{attribute 'qualified_only'}
VAR_GLOBAL
    stUnknownState: DUT_PositionState := (sName := 'Unknown');
    stInvalidState: DUT_PositionState;
END_VAR

(* stored: Version 1.1.0.1, ProductVersion 3.1.4022.18
   GVL MOTION_GVL: Id {7b3cfad1-1f36-4ed6-b576-62277c19b2b2} *)
